// TIA Portal V17 export
// export: Created 2023-02-26T22:28:46.0954072Z, ExportSetting WithDefaults, DisplayName Totally Integrated Automation Portal, DisplayVersion V17, DisplayName TIA Portal Openness, DisplayVersion V17, DisplayName TIA Portal Version Control Interface, DisplayVersion V17, DisplayName TIA Portal Test Suite Advanced, DisplayVersion V17, DisplayName STEP 7 Professional, DisplayVersion V17, DisplayName SIMATIC Energy Suite, DisplayVersion V17, DisplayName STEP 7 Safety, DisplayVersion V17, DisplayName WinCC Professional, DisplayVersion V17
FUNCTION_BLOCK "ERR_ChangeMode"   // FB10, LAD
{ S7_Optimized_Access := 'TRUE' }
VERSION : 0.1
// stored: AutoNumber true, IsIECCheckEnabled false, IsRetainMemResEnabled false, MemoryReserve 100, SetENOAutomatically false, UDAEnableTagReadback false
   VAR_INPUT
      StartLine : Bool;
      StopLine : Bool;
      ModeAuto : Bool;
      ModeManual : Bool;
      ResetButton : Bool;
      AlarmSiren : Bool;
      FirstScan : Bool;
   END_VAR
   VAR_OUTPUT
      Error : Bool;
   END_VAR
   VAR
      S1 : Bool;
      S2 : Bool;
      S3 : Bool;
      S4 : Bool;
      S5 : Bool;
      P_ResetButton : Bool;
   END_VAR
   VAR_TEMP   // added for the SCL form of the ladder/FBD networks
      _w1 : Bool;
   END_VAR
BEGIN

REGION Network 1
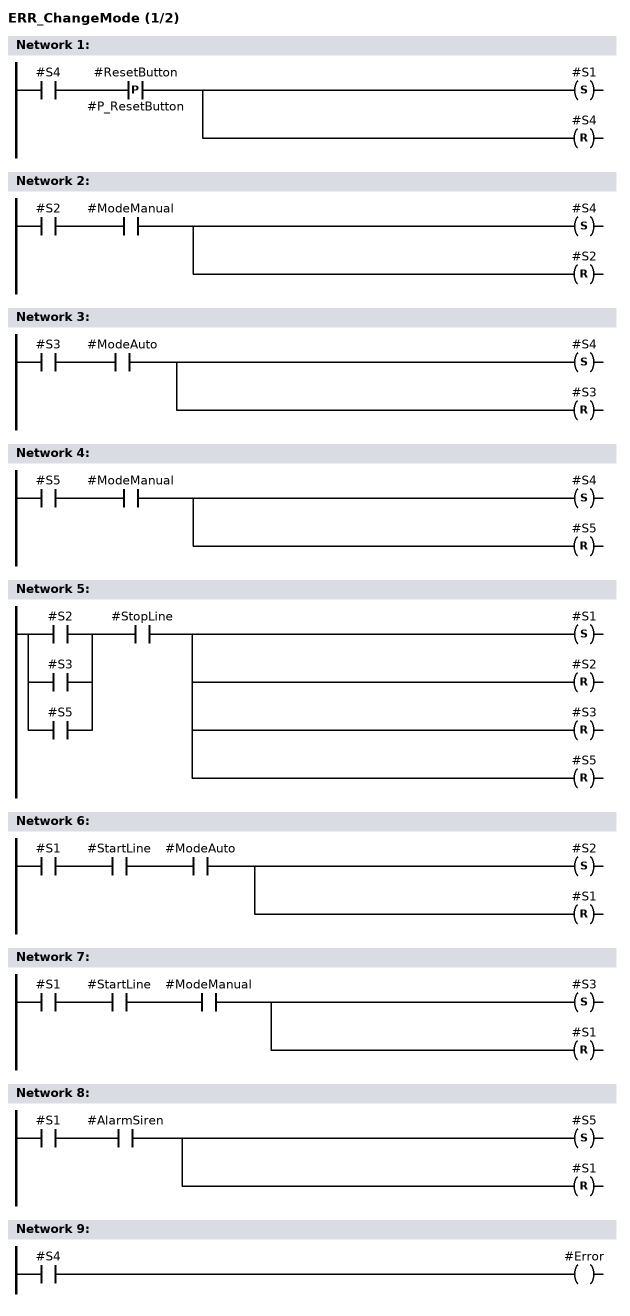
   RUNG wire#powerrail
      Contact( #S4 )
      P_Contact(operand := #ResetButton, bit := #P_ResetButton)
      wire#w1
      S_Coil( #S1 )
   END_RUNG
   RUNG wire#w1
      R_Coil( #S4 )
   END_RUNG
   // the same network as SCL:
   #_w1 := #S4 AND #ResetButton AND NOT #P_ResetButton;   // rising edge of #ResetButton
   #P_ResetButton := #ResetButton;
   IF #_w1 THEN
       #S1 := TRUE;
       #S4 := FALSE;
   END_IF;
END_REGION

REGION Network 2
   RUNG wire#powerrail
      Contact( #S2 )
      Contact( #ModeManual )
      wire#w1
      S_Coil( #S4 )
   END_RUNG
   RUNG wire#w1
      R_Coil( #S2 )
   END_RUNG
   // the same network as SCL:
   IF #S2 AND #ModeManual THEN
       #S4 := TRUE;
       #S2 := FALSE;
   END_IF;
END_REGION

REGION Network 3
   RUNG wire#powerrail
      Contact( #S3 )
      Contact( #ModeAuto )
      wire#w1
      S_Coil( #S4 )
   END_RUNG
   RUNG wire#w1
      R_Coil( #S3 )
   END_RUNG
   // the same network as SCL:
   IF #S3 AND #ModeAuto THEN
       #S4 := TRUE;
       #S3 := FALSE;
   END_IF;
END_REGION

REGION Network 4
   RUNG wire#powerrail
      Contact( #S5 )
      Contact( #ModeManual )
      wire#w1
      S_Coil( #S4 )
   END_RUNG
   RUNG wire#w1
      R_Coil( #S5 )
   END_RUNG
   // the same network as SCL:
   IF #S5 AND #ModeManual THEN
       #S4 := TRUE;
       #S5 := FALSE;
   END_IF;
END_REGION

REGION Network 5
   RUNG wire#powerrail
      Contact( #S2 )
      wire#w1
      Contact( #StopLine )
      wire#w2
      S_Coil( #S1 )
   END_RUNG
   RUNG wire#powerrail
      Contact( #S3 )
   END_RUNG wire#w1
   RUNG wire#powerrail
      Contact( #S5 )
   END_RUNG wire#w1
   RUNG wire#w2
      R_Coil( #S2 )
   END_RUNG
   RUNG wire#w2
      R_Coil( #S3 )
   END_RUNG
   RUNG wire#w2
      R_Coil( #S5 )
   END_RUNG
   // the same network as SCL:
   IF (#S2 OR #S3 OR #S5) AND #StopLine THEN #S1 := TRUE; END_IF;
   #_w1 := (#S2 OR #S3 OR #S5) AND #StopLine;
   IF #_w1 THEN
       #S2 := FALSE;
       #S3 := FALSE;
       #S5 := FALSE;
   END_IF;
END_REGION

REGION Network 6
   RUNG wire#powerrail
      Contact( #S1 )
      Contact( #StartLine )
      Contact( #ModeAuto )
      wire#w1
      S_Coil( #S2 )
   END_RUNG
   RUNG wire#w1
      R_Coil( #S1 )
   END_RUNG
   // the same network as SCL:
   IF #S1 AND #StartLine AND #ModeAuto THEN
       #S2 := TRUE;
       #S1 := FALSE;
   END_IF;
END_REGION

REGION Network 7
   RUNG wire#powerrail
      Contact( #S1 )
      Contact( #StartLine )
      Contact( #ModeManual )
      wire#w1
      S_Coil( #S3 )
   END_RUNG
   RUNG wire#w1
      R_Coil( #S1 )
   END_RUNG
   // the same network as SCL:
   IF #S1 AND #StartLine AND #ModeManual THEN
       #S3 := TRUE;
       #S1 := FALSE;
   END_IF;
END_REGION

REGION Network 8
   RUNG wire#powerrail
      Contact( #S1 )
      Contact( #AlarmSiren )
      wire#w1
      S_Coil( #S5 )
   END_RUNG
   RUNG wire#w1
      R_Coil( #S1 )
   END_RUNG
   // the same network as SCL:
   IF #S1 AND #AlarmSiren THEN
       #S5 := TRUE;
       #S1 := FALSE;
   END_IF;
END_REGION

REGION Network 9
   RUNG wire#powerrail
      Contact( #S4 )
      Coil( #Error )
   END_RUNG
   // the same network as SCL:
   #Error := #S4;
END_REGION

REGION Network 10
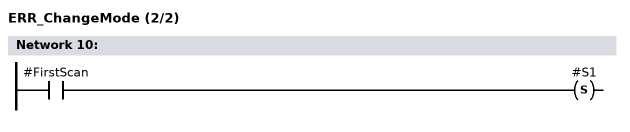
   RUNG wire#powerrail
      Contact( #FirstScan )
      S_Coil( #S1 )
   END_RUNG
   // the same network as SCL:
   IF #FirstScan THEN #S1 := TRUE; END_IF;
END_REGION
END_FUNCTION_BLOCK
